FUNCTION_BLOCK MPC_MEDIAN_FILTER_9 (* Deterministic 9-sample rolling median for the raw-count MPC model coordinate *)
  (* Standard: 61499-2 *)
  (* Version 1.0, 2026-08-10, Guilherme *)
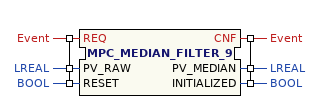
  EVENT_INPUT
    REQ WITH PV_RAW, RESET; (* Process one new raw level sample *)
  END_EVENT
  EVENT_OUTPUT
    CNF WITH PV_MEDIAN, INITIALIZED; (* Median value updated *)
  END_EVENT
  VAR_INPUT
    PV_RAW : LREAL; (* Current unfiltered raw level count *)
    RESET : BOOL; (* Refill the complete 9-sample buffer with the current input *)
  END_VAR
  VAR_OUTPUT
    PV_MEDIAN : LREAL; (* Median of the most recent 9 samples *)
    INITIALIZED : BOOL; (* Filter buffer has deterministic initialized content *)
  END_VAR
  VAR
    initialized_internal : BOOL := FALSE;
    v0 : LREAL := 0.0;
    v1 : LREAL := 0.0;
    v2 : LREAL := 0.0;
    v3 : LREAL := 0.0;
    v4 : LREAL := 0.0;
    v5 : LREAL := 0.0;
    v6 : LREAL := 0.0;
    v7 : LREAL := 0.0;
    v8 : LREAL := 0.0;
    s0 : LREAL := 0.0;
    s1 : LREAL := 0.0;
    s2 : LREAL := 0.0;
    s3 : LREAL := 0.0;
    s4 : LREAL := 0.0;
    s5 : LREAL := 0.0;
    s6 : LREAL := 0.0;
    s7 : LREAL := 0.0;
    s8 : LREAL := 0.0;
    swap_value : LREAL := 0.0;
  END_VAR
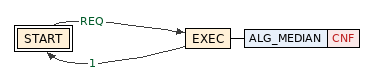
  EC_STATES
    START;
    EXEC : ALG_MEDIAN -> CNF;
  END_STATES
  EC_TRANSITIONS
    START TO EXEC := REQ;
    EXEC TO START := 1;
  END_TRANSITIONS
  ALGORITHM ALG_MEDIAN IN ST: (* Shift the sample history and compute an exact median using a fixed compare-swap network *)
IF RESET OR NOT initialized_internal THEN
    v0 := PV_RAW;
    v1 := PV_RAW;
    v2 := PV_RAW;
    v3 := PV_RAW;
    v4 := PV_RAW;
    v5 := PV_RAW;
    v6 := PV_RAW;
    v7 := PV_RAW;
    v8 := PV_RAW;
    initialized_internal := TRUE;
ELSE
    v0 := v1;
    v1 := v2;
    v2 := v3;
    v3 := v4;
    v4 := v5;
    v5 := v6;
    v6 := v7;
    v7 := v8;
    v8 := PV_RAW;
END_IF;

s0 := v0;
s1 := v1;
s2 := v2;
s3 := v3;
s4 := v4;
s5 := v5;
s6 := v6;
s7 := v7;
s8 := v8;

IF s0 > s1 THEN
    swap_value := s0;
    s0 := s1;
    s1 := swap_value;
END_IF;
IF s2 > s3 THEN
    swap_value := s2;
    s2 := s3;
    s3 := swap_value;
END_IF;
IF s4 > s5 THEN
    swap_value := s4;
    s4 := s5;
    s5 := swap_value;
END_IF;
IF s6 > s7 THEN
    swap_value := s6;
    s6 := s7;
    s7 := swap_value;
END_IF;
IF s1 > s2 THEN
    swap_value := s1;
    s1 := s2;
    s2 := swap_value;
END_IF;
IF s3 > s4 THEN
    swap_value := s3;
    s3 := s4;
    s4 := swap_value;
END_IF;
IF s5 > s6 THEN
    swap_value := s5;
    s5 := s6;
    s6 := swap_value;
END_IF;
IF s7 > s8 THEN
    swap_value := s7;
    s7 := s8;
    s8 := swap_value;
END_IF;
IF s0 > s1 THEN
    swap_value := s0;
    s0 := s1;
    s1 := swap_value;
END_IF;
IF s2 > s3 THEN
    swap_value := s2;
    s2 := s3;
    s3 := swap_value;
END_IF;
IF s4 > s5 THEN
    swap_value := s4;
    s4 := s5;
    s5 := swap_value;
END_IF;
IF s6 > s7 THEN
    swap_value := s6;
    s6 := s7;
    s7 := swap_value;
END_IF;
IF s1 > s2 THEN
    swap_value := s1;
    s1 := s2;
    s2 := swap_value;
END_IF;
IF s3 > s4 THEN
    swap_value := s3;
    s3 := s4;
    s4 := swap_value;
END_IF;
IF s5 > s6 THEN
    swap_value := s5;
    s5 := s6;
    s6 := swap_value;
END_IF;
IF s7 > s8 THEN
    swap_value := s7;
    s7 := s8;
    s8 := swap_value;
END_IF;
IF s0 > s1 THEN
    swap_value := s0;
    s0 := s1;
    s1 := swap_value;
END_IF;
IF s2 > s3 THEN
    swap_value := s2;
    s2 := s3;
    s3 := swap_value;
END_IF;
IF s4 > s5 THEN
    swap_value := s4;
    s4 := s5;
    s5 := swap_value;
END_IF;
IF s6 > s7 THEN
    swap_value := s6;
    s6 := s7;
    s7 := swap_value;
END_IF;
IF s1 > s2 THEN
    swap_value := s1;
    s1 := s2;
    s2 := swap_value;
END_IF;
IF s3 > s4 THEN
    swap_value := s3;
    s3 := s4;
    s4 := swap_value;
END_IF;
IF s5 > s6 THEN
    swap_value := s5;
    s5 := s6;
    s6 := swap_value;
END_IF;
IF s7 > s8 THEN
    swap_value := s7;
    s7 := s8;
    s8 := swap_value;
END_IF;
IF s0 > s1 THEN
    swap_value := s0;
    s0 := s1;
    s1 := swap_value;
END_IF;
IF s2 > s3 THEN
    swap_value := s2;
    s2 := s3;
    s3 := swap_value;
END_IF;
IF s4 > s5 THEN
    swap_value := s4;
    s4 := s5;
    s5 := swap_value;
END_IF;
IF s6 > s7 THEN
    swap_value := s6;
    s6 := s7;
    s7 := swap_value;
END_IF;
IF s1 > s2 THEN
    swap_value := s1;
    s1 := s2;
    s2 := swap_value;
END_IF;
IF s3 > s4 THEN
    swap_value := s3;
    s3 := s4;
    s4 := swap_value;
END_IF;
IF s5 > s6 THEN
    swap_value := s5;
    s5 := s6;
    s6 := swap_value;
END_IF;
IF s7 > s8 THEN
    swap_value := s7;
    s7 := s8;
    s8 := swap_value;
END_IF;
IF s0 > s1 THEN
    swap_value := s0;
    s0 := s1;
    s1 := swap_value;
END_IF;
IF s2 > s3 THEN
    swap_value := s2;
    s2 := s3;
    s3 := swap_value;
END_IF;
IF s4 > s5 THEN
    swap_value := s4;
    s4 := s5;
    s5 := swap_value;
END_IF;
IF s6 > s7 THEN
    swap_value := s6;
    s6 := s7;
    s7 := swap_value;
END_IF;

PV_MEDIAN := s4;
INITIALIZED := initialized_internal;
  END_ALGORITHM
END_FUNCTION_BLOCK
